PROGRAM prgEMS
VAR
	EMS					: FB_EMS;			//{#lynus.ag#()}
	iMassageEMS			: INT;				//{#lynus.ag#()}
	fbreboot			: NT_Reboot;
END_VAR

EMS(
	bEnable:= , 
	diNrOfEM_IN_ECS:= , 
	stSetupEMS:= , 
	eOperationMode:= ,
	eSpeedModeBackendController:= E_SpeedModeBackendController_EMS.eSlow, 
	eSpeedModeLocalController:= E_SpeedModeLocalController_EMS.eBalanced,
	eMessageEMS=> , 
	bStateEnable=> , 
	bStateAllowChrgFromGrid=> , 
	bMissingPowerData=> , 
	bSurplusAvailable=> , 
	bActivateHP=> , 
	bControllingState=> , 
	byProgress=> , 
	diNrOfEMS_OUT=> , 
	rHeartbeat=> , 
	rErrorWarning=> , 
	rEnergyOptReady=> , 
	rNewBattPower=> , 
	arrMinPrioReached=> , 
	arrMaxPrioReached=> );
	
iMassageEMS := ems.eMessageEMS;

fbreboot(
	NETID:= , 
	DELAY:= , 
	START:= , 
	TMOUT:= , 
	BUSY=> , 
	ERR=> , 
	ERRID=> );

END_PROGRAM

(* stored: Version 1.1.0.1, ProductVersion 3.1.4024.9
   POU prgEMS: Id {cd09de00-7d0c-4acf-aa0f-0b56eaa0eb3f}, SpecialFunc None *)
